// Recipe for the 21.101 machine
TYPE Recipe_21_101_t :
STRUCT
    linearAxis : ARRAY[0..LinearAxis_e._max - 1] OF LinearMotionMan_Config_t;
    st110      : ST110_Recipe_t;
    st115      : ST115_Recipe_t;
END_STRUCT
END_TYPE

(* stored: Version 1.1.0.1, ProductVersion 3.1.4024.6
   DUT Recipe_21_101_t: Id {44f7e314-df6d-4947-97da-ae80be0f8d1d} *)
